{attribute 'GeneratedUsingTerminal: EPP1322-0001-0017'}
{attribute addProperty BoxType "EPP1322-0001-0017"}
{attribute addProperty Id "RC60_AB1_EPP1008_0001EPP1008_78E8D3DD12RC60_AB2_EPP1008_0001EPP1008_78E8D3DD12RC60_AB6_EPP1008_0001EPP1008_78E8D3DD12RC60_AB3_EPP1008_0001EPP1008_78E8D3DD12RC60_AB4_EPP1008_0001EPP1008_78E8D3DD12RC60_AB7_EPP1008_0001EPP1008_78E8D3DD12RC60_AB9_EPP1008_0001EPP1008_78E8D3DD12RC60_AB10_EPP1008_0001EPP1008_78E8D3DD12RC60_AB8_EPP1008_0001EPP1008_78E8D3DD12RC60_AB5_EPP1008_0001EPP1008_78E8D3DD12"}
{attribute addProperty CRC "2154990392"}
{attribute addProperty Size "120"}
{attribute addProperty Name "RC60_EPP (EPP1322-0001)"}
TYPE RC60_EPP_EPP1322_0001_80728B38 EXTENDS EPP1322_1FC0878B : 
STRUCT
    {attribute addProperty Name "RC60_AB1 (EPP1008-0001)"}
    {attribute addProperty PreviousPort "RC60_EPP (EPP1322-0001) : D"}
    {attribute addProperty SyncUnit "C60"}
    RC60_AB1_EPP1008_0001 : EPP1008_78E8D3DD;
    {attribute addProperty Name "RC60_AB2 (EPP1008-0001)"}
    {attribute addProperty PreviousPort "RC60_AB1 (EPP1008-0001) : B"}
    {attribute addProperty SyncUnit "C60"}
    RC60_AB2_EPP1008_0001 : EPP1008_78E8D3DD;
    {attribute addProperty Name "RC60_AB6 (EPP1008-0001)"}
    {attribute addProperty PreviousPort "RC60_AB2 (EPP1008-0001) : B"}
    {attribute addProperty SyncUnit "C60"}
    RC60_AB6_EPP1008_0001 : EPP1008_78E8D3DD;
    {attribute addProperty Name "RC60_AB3 (EPP1008-0001)"}
    {attribute addProperty PreviousPort "RC60_AB6 (EPP1008-0001) : B"}
    {attribute addProperty SyncUnit "C60"}
    RC60_AB3_EPP1008_0001 : EPP1008_78E8D3DD;
    {attribute addProperty Name "RC60_AB4 (EPP1008-0001)"}
    {attribute addProperty PreviousPort "RC60_AB3 (EPP1008-0001) : B"}
    {attribute addProperty SyncUnit "C60"}
    RC60_AB4_EPP1008_0001 : EPP1008_78E8D3DD;
    {attribute addProperty Name "RC60_AB7 (EPP1008-0001)"}
    {attribute addProperty PreviousPort "RC60_EPP (EPP1322-0001) : B"}
    {attribute addProperty SyncUnit "C60"}
    RC60_AB7_EPP1008_0001 : EPP1008_78E8D3DD;
    {attribute addProperty Name "RC60_AB9 (EPP1008-0001)"}
    {attribute addProperty PreviousPort "RC60_AB7 (EPP1008-0001) : B"}
    {attribute addProperty SyncUnit "C60"}
    RC60_AB9_EPP1008_0001 : EPP1008_78E8D3DD;
    {attribute addProperty Name "RC60_AB10 (EPP1008-0001)"}
    {attribute addProperty PreviousPort "RC60_AB9 (EPP1008-0001) : B"}
    {attribute addProperty SyncUnit "C60"}
    RC60_AB10_EPP1008_0001 : EPP1008_78E8D3DD;
    {attribute addProperty Name "RC60_AB8 (EPP1008-0001)"}
    {attribute addProperty PreviousPort "RC60_AB10 (EPP1008-0001) : B"}
    {attribute addProperty SyncUnit "C60"}
    RC60_AB8_EPP1008_0001 : EPP1008_78E8D3DD;
    {attribute addProperty Name "RC60_AB5 (EPP1008-0001)"}
    {attribute addProperty PreviousPort "RC60_AB8 (EPP1008-0001) : B"}
    {attribute addProperty SyncUnit "C60"}
    RC60_AB5_EPP1008_0001 : EPP1008_78E8D3DD;
END_STRUCT
END_TYPE

(* stored: Version 1.2.0.0, ProductVersion 3.1.4024.11
   DUT RC60_EPP_EPP1322_0001_80728B38: Id {2ee0b774-bf99-0565-2403-77bfa6bda29d} *)
